(* PLC project Tc2_Utilities.F_BIGTYPE Demo, tc3-libraries-kb TwinCAT 3.1 *)
(* stored: creationDateTime 2026-05-11T00:00:00, modificationDateTime 2026-05-11T00:00:00 *)

TYPE ST_Recipe : STRUCT
  nRecipeId : UDINT;
  fTargetTempC : LREAL;
  tHoldDuration : TIME;
  bIsActive : BOOL;
END_STRUCT;
END_TYPE

PROGRAM P_Demo_F_BIGTYPE
  VAR
    stCurrentRecipe : ST_Recipe;  (* 当前配方 *)
    argRecipe : T_Arg;  (* 配方打包后的 T_Arg *)
    bPackRecipe : BOOL;  (* 在线置 TRUE 触发一次打包 *)
  END_VAR

            // ============================================================
// Tc2_Utilities.F_BIGTYPE 演示程序
// ============================================================
// 场景：把整段配方结构体作为一个 T_Arg 送给 EventLogger 当报警上下文。
// 价值：结构体没有专用 F_<TYPE>，本函数按字节打包；下游靠 cbLen 取整段。
// 验证：在线写 stCurrentRecipe.nRecipeId := 7、bPackRecipe := TRUE；
//       下一周期 argRecipe.cbLen 应等于 SIZEOF(stCurrentRecipe)，argRecipe.pData <> 0。
// ============================================================

IF bPackRecipe THEN
    // 用 ADR + SIZEOF 把整个结构体打包，eType 自动选 BIGTYPE 枚举
    argRecipe := F_BIGTYPE(pData := ADR(stCurrentRecipe),
                           cbLen := SIZEOF(stCurrentRecipe));
    bPackRecipe := FALSE;
END_IF;

          
END_PROGRAM
